(* IEC 61131-3 sources: mastertool-rankine-bridge/tests/indexer/fixtures/sample_export/objects/application_gvl_2__GvlAmbiguaSintetica, 1 file *)

(* ---- declaration.st ---- *)
VAR_GLOBAL
    DG_Contador : DINT;
    GA_ValorSintetico : INT;
END_VAR
